{attribute 'qualified_only'}
{attribute 'strict'}
TYPE E_ReloadRoundBelt_PlaceArea :
(
	Undefined := 0,
	RoundBelt
)UINT;
END_TYPE

(* stored: Version 1.1.0.1, ProductVersion 3.1.4024.13
   DUT E_ReloadRoundBelt_PlaceArea: Id {ff50fd77-b40a-4292-a7bf-55cd2de710c1} *)
